FUNCTION_BLOCK SC_BeltConveyors EXTENDS FB_Chain
VAR_INPUT
	bExecute : BOOL;
	bAllPartsPresent : BOOL;
END_VAR
VAR_OUTPUT
END_VAR
VAR
	aBeltConveyors : ARRAY[1..2] OF BeltConveyor;
	fbCounterSensor : Sensor;
	i : INT;
	uiPackageCounter : UINT;
	fbTrig : R_TRIG;
	
END_VAR

SUPER^();
fbCounterSensor();
fbTrig(CLK := fbCounterSensor.bSignal);
IF fbTrig.Q
THEN
	uiPackageCounter := uiPackageCounter + 1;
END_IF
FOR i := 1 TO (eMaxNumBeltConveyors - 1)
DO
	
	aBeltConveyors[i]();

END_FOR

METHOD PROTECTED Busy : BOOL
VAR_INPUT
END_VAR
VAR
	iStepCondition : I_StepCondition;
END_VAR
fbStepWorkerBusy();

CASE fbStepWorkerBusy.uiStep OF

	eBusySCStart: 
		THIS^.aBeltConveyors[eBeltConveyorEntrance].On();
		
		fbStepWorkerBusy.mNextStep(10);
		
	10:
		//As Soon as the first package reaches the counter sensor
		//the second floor of the palletizer is informed
		//consequently the second floor of the palletizer will go in busy mode.
		IF uiPackageCounter = 1
		THEN
			THIS^.aBeltConveyors[eBeltConveyorUpwards].On();
			
			fbStepWorkerBusy.mNextStep(15);
		END_IF
		
	15:
		IF uiPackageCounter = 3
		THEN
			uiPackageCounter := 0;
			fbStepWorkerBusy.mNextStep(20);
		END_IF
	20:
		fbStepWorkerBusy
				.mSetTimer(T#1s)
				.mNextStep(30);
	30:
		THIS^.aBeltConveyors[eBeltConveyorEntrance].Off();
		IF bAllPartsPresent
		THEN
			THIS^.aBeltConveyors[eBeltConveyorUpwards].Off();
			Done();
			fbStepWorkerBusy.mNextStep(0);
		END_IF
		
	40:
	
		
		(*
		//At start we check how many packages have passed the fbCounterSensor
		IF uiPackageCounter < 3
		THEN
		
			//activate the conveyors
			fbStepWorkerBusy.mNextStep(eStartEntranceConveyor);
			
		ELSIF uiPackageCounter = 3
		 AND NOT ioPalletizer.bAllPartsPresent
		 AND aBeltConveyors[eBeltConveyorEntrance].bStart
		THEN
 			//A package needs to reach the palletizer or a sensor is malfunctioning		
			fbStepWorkerBusy
				.mSetTimer(T#1s)
				.mNextStep(eStopEntranceConveyor);
				
		ELSIF uiPackageCounter = 3
		 AND ioPalletizer.bAllPartsPresent
	 	THEN
			//Execute the Palletizer
			uiPackageCounter := 0;
			aBeltConveyors[eBeltConveyorUpwards].Off();
			fbStepWorkerBusy.mNextStep(eWaitForPalletizer);
		ELSIF uiPackageCounter > 3
		THEN
			//Error
		END_IF
		
	eStartEntranceConveyor:
		
		aBeltConveyors[eBeltConveyorEntrance].On();
		fbStepWorkerBusy.mAddCondition(fbCounterSensor.getSignal);
		fbStepWorkerBusy.mNextStep(eStartUpwardsConveyor);

	eStartUpwardsConveyor:
	
		
		aBeltConveyors[eBeltConveyorUpwards].On();
		fbStepWorkerBusy.mNextStep(eExecutePalletizer);
			 
	eExecutePalletizer:
		 
		ioPalletizer.Execute();	
		fbStepWorkerBusy.mNextStep(eBusySCStart);
	
	eStopEntranceConveyor:
		aBeltConveyors[eBeltConveyorEntrance].Off();
		fbStepWorkerBusy.mNextStep(eExecutePalletizer);
		
	eWaitForPalletizer:
	
		 fbStepWorkerBusy.mAddCondition(ioPalletizer.getDoneCycle);
		 fbStepWorkerBusy.mNextStep(eBusySCStart);
		 
	eSignalError:
	
		fbStepWorkerBusy.mNextStep(eBusySCStart);
		Fault();	
		*)	
END_CASE
END_METHOD

METHOD PROTECTED  Error : BOOL
VAR_INPUT
END_VAR
VAR
	i : INT;
END_VAR
FOR i := 1 TO 3 
DO

	aBeltConveyors[i].Off();
	
END_FOR
END_METHOD

METHOD PROTECTED  Idle : BOOL
VAR_INPUT
END_VAR
END_METHOD

METHOD PROTECTED  Init : BOOL
VAR_INPUT
END_VAR
Start();
END_METHOD

METHOD PROTECTED  Prepare : BOOL
VAR_INPUT
END_VAR
END_METHOD

METHOD PROTECTED  Ready : BOOL
VAR_INPUT
END_VAR
fbStepWorkerReady();
CASE fbStepWorkerReady.uiStep OF
	
	0: 
	
		IF bExecute THEN
			fbStepWorkerReady.mNextStep(10);
		END_IF
		
	10:
	
		IF rChainController
			.releaseCheck(THIS^)
			.releaseFromChain(sChainReleasing := 'scSecondFloor', THIS^)
			.releaseResult(THIS^) 
		THEN
			Execute();
			rChainController.releaseForChain('scSecondFloor', THIS^);		
			fbStepWorkerReady.mNextStep(0);
		END_IF
	
		
	
END_CASE
END_METHOD

METHOD PROTECTED  Waiting : BOOL
VAR_INPUT
END_VAR
END_METHOD

END_FUNCTION_BLOCK

(* stored: Version 1.1.0.1, ProductVersion 3.1.4024.2
   POU SC_BeltConveyors: Id {dd4c126b-b2e6-47bc-929b-e6a020fb882e}, SpecialFunc None
   Method Busy: Id {3dac21d8-7436-41fb-b699-d5668543a826}
   Method Error: Id {1094dc30-0ff4-41f2-a537-8aae3d176300}
   Method Idle: Id {390b6e72-0a77-4967-a4a7-b01388167acc}
   Method Init: Id {6c991035-b97c-4a4c-b1ba-d7201673aa97}
   Method Prepare: Id {d29b2afb-d034-4d97-96dc-e776605b5e25}
   Method Ready: Id {3f1e5b29-9a5c-4009-8817-888b67885389}
   Method Waiting: Id {e15a1ec5-6f67-48c4-98c6-44a18b3ede63} *)
